{attribute 'no_explicit_call' := 'Body contains no logic, calling methods only allowed.'}
FUNCTION_BLOCK INTERNAL FB_Wildcards

// Matches any number of characters. You can use the asterisk (*) anywhere in a character string.
// Example: wh* finds what, white, and why, but not awhile or watch.
PROPERTY Asterisk : ZigaLibs_Core.T_Char
GET
Asterisk := '*';
END_GET
END_PROPERTY

// Matches a single alphabet in a specific position.
// Example: b?ll finds ball, bell, and bill.
PROPERTY QuestionMark : ZigaLibs_Core.T_Char
GET
QuestionMark := '?';
END_GET
END_PROPERTY

END_FUNCTION_BLOCK

(* stored: Version 1.1.0.1, ProductVersion 3.1.4024.14
   POU FB_Wildcards: Id {77d495e7-1020-0e62-286d-5845201f3faa}, SpecialFunc None
   Property Asterisk: Id {a731c642-d997-00cc-3f9a-139dca7bb981}
   Get Get: Id {4eb674a2-9788-0d26-0543-fbcf2a29ec9e}
   Property QuestionMark: Id {f79dd64b-cf89-0e1e-0705-63c0f68a78a5}
   Get Get: Id {88a4cb75-9979-0e08-2a04-cf775f91b985} *)
